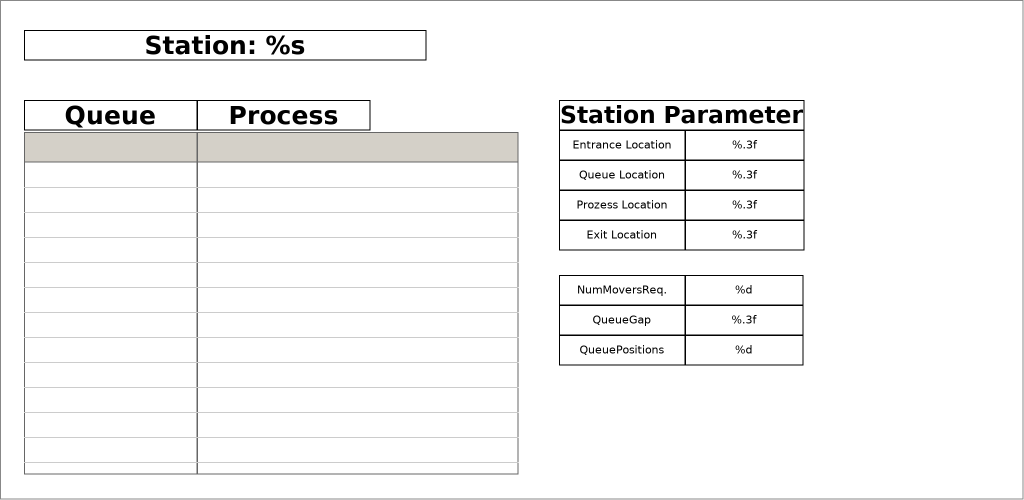
VISUALIZATION VI_StationSub  // 1024x500
    Rectangle (24,30 402x30), "Station: %s", text variable: GVL_XPlanarVisuDiag.sStationName
    Rectangle (24,100 173x30), "Queue"
    Rectangle (197,100 173x30), "Process"
    Table (197,132 321x342), data array: GVL_StationVisu.aMoverInSequence
        p1128707560: GVL_XPlanarVisuDiag.gcnMaxMoverInStation
        p3854506369: GVL_StationVisu.aMoverInSequence[INDEX].nMover
        p1892666644: GVL_StationVisu.aMoverInSequence[INDEX].nSequence
        p2232123230: GVL_XPlanarVisuDiag.aMoverInSequence[INDEX].nMover
        p511219082: GVL_XPlanarVisuDiag.aMoverInSequence[INDEX].nSequence
    Table (24,132 173x342), data array: GVL_XPlanarVisuDiag.aMoverInQueue
        p1128707560: GVL_XPlanarVisuDiag.gcnMaxMoverInStation
        p3854506369: GVL_XPlanarVisuDiag.aMoverInQueue[INDEX]
    Rectangle (559,100 245x30), "Station Parameter"
    Rectangle (559,130 126x30), "Entrance Location"
    Rectangle (559,160 126x30), "Queue Location"
    Rectangle (559,190 126x30), "Prozess Location"
    Rectangle (559,220 126x30), "Exit Location"
    Rectangle (559,275 126x30), "NumMoversReq."
    Rectangle (559,305 126x30), "QueueGap"
    Rectangle (559,335 126x30), "QueuePositions"
    Rectangle (685,130 119x30), "%.3f", text variable: GVL_XPlanarVisuDiag.stStationConfig.fEntranceLocation
    Rectangle (685,160 119x30), "%.3f", text variable: GVL_XPlanarVisuDiag.stStationConfig.fQueueLocation
    Rectangle (685,190 119x30), "%.3f", text variable: GVL_XPlanarVisuDiag.stStationConfig.fProzessLocation
    Rectangle (685,220 119x30), "%.3f", text variable: GVL_XPlanarVisuDiag.stStationConfig.fExitLocation
    Rectangle (685,275 118x30), "%d", text variable: GVL_XPlanarVisuDiag.stStationConfig.nNumMoversRequired
    Rectangle (685,305 118x30), "%.3f", text variable: GVL_XPlanarVisuDiag.stStationConfig.fQueueGap
    Rectangle (685,335 118x30), "%d", text variable: GVL_XPlanarVisuDiag.stStationConfig.nNumQueuePositions
END_VISUALIZATION

(* stored: Version 1.1.0.1, ProductVersion 3.1.4024.9
   Visu VI_StationSub: Id {1603bfa7-1fea-48b8-aabd-a82c7f7961f3} *)
